// TIA Portal V16 export
// export: Created 2024-04-23T10:21:57.3163423Z, ExportSetting WithDefaults, DisplayName Totally Integrated Automation Portal, DisplayVersion V16 Update 5, DisplayName TIA Portal Version Control Interface, DisplayVersion V16 Update 2, DisplayName TIA Portal Openness, DisplayVersion V16 Update 5, DisplayName TIA Portal Teamcenter Gateway, DisplayVersion V16, DisplayName SINAMICS Startdrive Advanced, DisplayVersion V16, DisplayName SINAMICS Startdrive G130, G150, S120, S150, SINAMICS MV, S210, DisplayVersion V16, DisplayName SINAMICS Startdrive G110M, G120, G120C, G120D, G120P, DisplayVersion V16, DisplayName STEP 7 Professional, DisplayVersion V16 Update 5, DisplayName STEP 7 Safety, DisplayVersion V16, DisplayName WinCC UA Professional, DisplayVersion V16 Update 5
ORGANIZATION_BLOCK "Main"   // OB1, LAD, ProgramCycle
TITLE = "Main Program Sweep (Cycle)"
{ S7_Optimized_Access := 'TRUE' }
VERSION : 0.1
// stored: AutoNumber true, IsIECCheckEnabled false, SetENOAutomatically false
   VAR_INPUT
      Initial_Call : Bool;   // Initial call of this OB
      Remanence : Bool;   // =True, if remanent data are available
   END_VAR
BEGIN

REGION Network 1
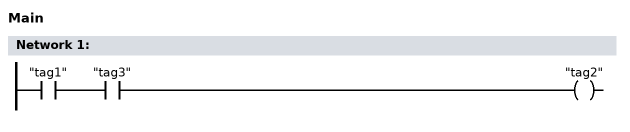
   RUNG wire#powerrail
      Contact( "tag1" )
      Contact( "tag3" )
      Coil( "tag2" )
   END_RUNG
   // the same network as SCL:
   "tag2" := "tag1" AND "tag3";
END_REGION
END_ORGANIZATION_BLOCK
